(* PLC project Tc2_Utilities.F_GenerateHashValue Demo, tc3-libraries-kb TwinCAT 3.1 *)
(* stored: creationDateTime 2026-05-10T19:00:00, modificationDateTime 2026-05-10T19:00:00 *)

PROGRAM P_Demo_F_GenerateHashValue
  VAR
    rResult : BOOL;  (* F_GenerateHashValue 返回值 *)
    bRun : BOOL;  (* 触发一次调用 *)
    sIn : STRING := 'hello';  (* 测试用本地变量 *)
    aHash : ARRAY[0..31] OF BYTE;  (* 测试用本地变量 *)
  END_VAR

            // ============================================================
// Tc2_Utilities.F_GenerateHashValue 演示程序（FUNCTION）
// ============================================================
// 验证步骤：
//   1. 引用 Tc2_Utilities
//   2. 编译 + 登录
//   3. 强制 bRun := TRUE 一个周期
//   4. 在线监视 rResult / 各 demo 变量
// ============================================================

IF bRun THEN
    rResult := F_GenerateHashValue(E_HashMode.eHashMode_SHA256, ADR(sIn), LEN(sIn), ADR(aHash), SIZEOF(aHash));
    bRun := FALSE;
END_IF;

          
END_PROGRAM
